INTERFACE ITF_PayloadHandler

END_INTERFACE

(* stored: Version 1.1.0.1
   Itf ITF_PayloadHandler: Id {bff43ede-aa01-4619-ab48-cbd1a274fc21} *)
